// TIA Portal V20 export
DATA_BLOCK "定位轴基本控制_取芯V90"   // DB6
// stored: InstanceOfName 定位轴基本控制, InstanceOfType FB
"定位轴基本控制"
   // VAR_INPUT
   //    轴号 : TO_PositioningAxis;
   //    使能 : Bool;
   //    回原 : Bool;
   //    回原模式 : Int;
   //    绝对定位 : Bool;
   //    相对定位 : Bool;
   //    暂停 : Bool;
   //    复位 : Bool;
   //    绝对位置 : Real;
   //    绝对速度 : Real;
   //    相对位置 : Real;
   //    相对速度 : Real;
   //    点动正转 : Bool;
   //    点动反转 : Bool;
   //    点动速度 : Real;
   // END_VAR
   // VAR_OUTPUT
   //    轴已启用 : Bool;
   //    使能错误 : Bool;
   //    回原完成 : Bool;
   //    回原错误 : Bool;
   //    绝对定位完成 : Bool;
   //    绝对定位错误 : Bool;
   //    相对定位完成 : Bool;
   //    相对定位错误 : Bool;
   //    点动中 : Bool;
   //    点动错误 : Bool;
   //    当前位置 : LReal;
   //    当前速度 : LReal;
   // END_VAR
   // VAR
   //    MC_Power_Instance { S7_SetPoint := 'True'} : MC_POWER;
   //    MC_Home_Instance { S7_SetPoint := 'True'} : MC_HOME;
   //    MC_MoveAbsolute_Instance { S7_SetPoint := 'True'} : MC_MOVEABSOLUTE;
   //    MC_MoveRelative_Instance { S7_SetPoint := 'True'} : MC_MOVERELATIVE;
   //    MC_Reset_Instance { S7_SetPoint := 'True'} : MC_RESET;
   //    MC_Halt_Instance { S7_SetPoint := 'True'} : MC_HALT;
   //    MC_MoveJog_Instance { S7_SetPoint := 'True'} : MC_MOVEJOG;
   // END_VAR
BEGIN
END_DATA_BLOCK
